(* IEC 61131-3 sources: eCockpitGit/test_project/src/%F%00 Library/%F%Common Functions/%F%Buffer/%POU%FB_FIFOArray, 5 files *)

(* ---- %METH%pushEnd.st ---- *)
//Releases the lock for getting the next index
// |**Version**|**Author**| **Date** |**Changes**
// | 1         | NSN      | 15-02-22 | Creation
METHOD pushEnd
(*%!%__DELIMITER__%!%*)
WHILE TRUE DO
	IF __COMPARE_AND_SWAP(ADR(S_block),0,1) THEN
		S_amount			:=		S_amount + 1;
		S_block				:=		0;
		EXIT;
	END_IF
END_WHILE
IF S_input < S_bufferSize - 1 THEN
	S_input					:=		S_input + S_startIndex + 1;
ELSE
	S_input					:=		S_startIndex;
END_IF

S_blockInput				:=		0;

(* ---- %METH%pushStart.st ---- *)
//Gets the next free index in the array, and locks inputs from other threads
//pushEnd must be called to free the thread lock made in this method
// |**Version**|**Author**| **Date** |**Changes**
// | 1         | NSN      | 15-02-22 | Creation
METHOD pushStart : BOOL
VAR_OUTPUT
	index		:DWORD;
END_VAR
(*%!%__DELIMITER__%!%*)
WHILE S_amount < S_bufferSize DO
	IF __COMPARE_AND_SWAP(ADR(S_blockInput),0,1) THEN
		IF S_amount = S_bufferSize THEN
			S_blockInput			:=		0;
			RETURN;
		END_IF
		IF S_input < S_bufferSize - 1 THEN
			index					:=		S_input + S_startIndex + 1;
		ELSE
			index					:=		S_startIndex;
		END_IF
		pushStart					:=		TRUE;
		RETURN;
	END_IF
END_WHILE

(* ---- %METH%setSize.st ---- *)
//Changes the size of the queue in a tread safe way
// |**Version**|**Author**| **Date** |**Changes**
// | 1         | NSN      | 15-02-22 | Creation
METHOD setSize
VAR_INPUT
	size		:DWORD;
END_VAR

(*%!%__DELIMITER__%!%*)
WHILE TRUE DO
	IF __COMPARE_AND_SWAP(ADR(S_blockInput),0,1) THEN
		WHILE TRUE DO
			IF __COMPARE_AND_SWAP(ADR(S_blockOutput),0,1) THEN
				S_bufferSize			:=		size;
				S_amount				:=		0;
				S_input					:=		0;
				S_output				:=		0;
				S_blockOutput			:=		0;
				S_blockInput			:=		0;
				RETURN;
			END_IF
		END_WHILE
	END_IF
END_WHILE

(* ---- %METH%unshiftEnd.st ---- *)
//Gets the oldest element from the buffer if there are any
// |**Version**|**Author**| **Date** |**Changes**
// | 1         | NSN      | 15-02-22 | Creation
METHOD unshiftEnd

(*%!%__DELIMITER__%!%*)
WHILE TRUE DO
	IF __COMPARE_AND_SWAP(ADR(S_block),0,1) THEN
		S_amount			:=		S_amount - 1;
		S_block				:=		0;
		EXIT;
	END_IF
END_WHILE
IF S_output < S_bufferSize - 1 THEN
	S_output				:=		S_output + S_startIndex + 1;
ELSE
	S_output				:=		S_startIndex;
END_IF

S_blockOutput				:=		0;

(* ---- %METH%unshiftStart.st ---- *)
//Gets the oldest element from the buffer if there are any
// |**Version**|**Author**| **Date** |**Changes**
// | 1         | NSN      | 15-02-22 | Creation
METHOD unshiftStart : BOOL
VAR_OUTPUT
	index		:DWORD;
END_VAR
(*%!%__DELIMITER__%!%*)
WHILE S_amount > 0 DO
	IF __COMPARE_AND_SWAP(ADR(S_blockOutput),0,1) THEN
		IF S_amount = 0 THEN
			S_blockOutput			:=		0;
			RETURN;
		END_IF
		IF S_output < S_bufferSize - 1 THEN
			index					:=		S_output + S_startIndex + 1;
		ELSE
			index					:=		S_startIndex;
		END_IF
		unshiftStart				:=		TRUE;
		RETURN;
	END_IF
END_WHILE
